% RSLogix 500 project UNTITLED_BAK061.RSS, saved by version 8.10.00.18 %
PROJECT "UNTITLED"    % processor: MicroLogix 1200 %

PROGRAM FILES
  LAD 2   19 rungs

DATA FILES
  O0 OUTPUT  4 elements
  I1 INPUT  4 elements
  S2 STATUS  66 elements
  B3 BINARY  1 elements
  T4 TIMER  7 elements
  C5 COUNTER  1 elements
  R6 CONTROL  1 elements
  N7 INTEGER  1 elements

LADDER 2
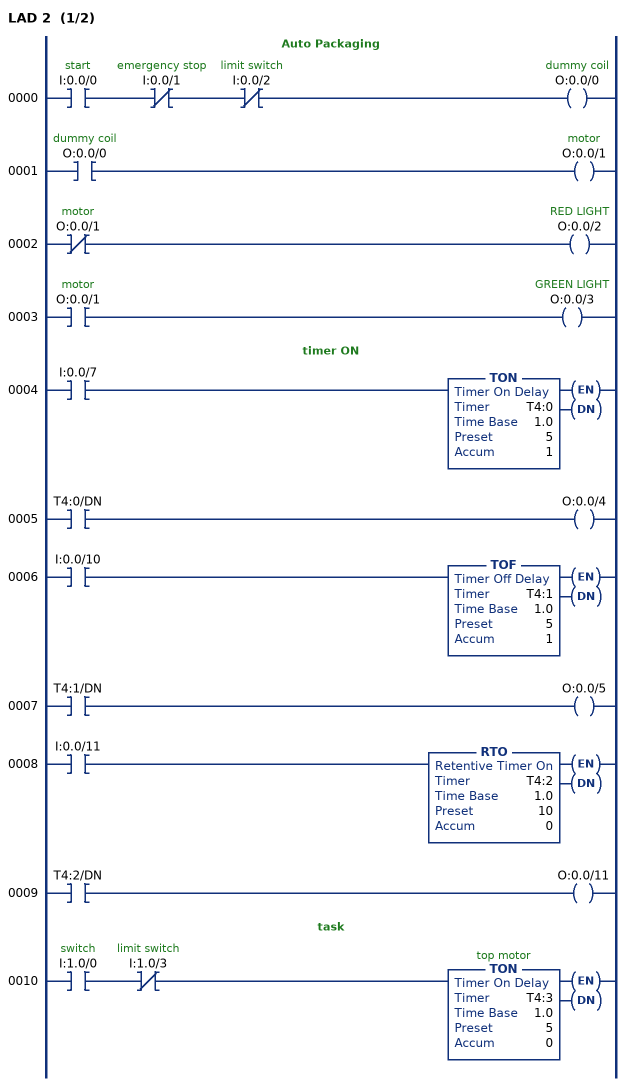
% Rung: 0 %
% TITLE: Auto Packaging %
SOR XIC I:0.0/0 XIO I:0.0/1 XIO I:0.0/2 OTE O:0.0/0 EOR
%   I:0.0/0  "start" %
%   I:0.0/1  "emergency stop" %
%   I:0.0/2  "limit switch" %
%   O:0.0/0  "dummy coil" %
% Rung: 1 %
SOR XIC O:0.0/0 OTE O:0.0/1 EOR
%   O:0.0/0  "dummy coil" %
%   O:0.0/1  "motor" %
% Rung: 2 %
SOR XIO O:0.0/1 OTE O:0.0/2 EOR
%   O:0.0/1  "motor" %
%   O:0.0/2  "RED LIGHT" %
% Rung: 3 %
SOR XIC O:0.0/1 OTE O:0.0/3 EOR
%   O:0.0/1  "motor" %
%   O:0.0/3  "GREEN LIGHT" %
% Rung: 4 %
% TITLE: timer ON %
SOR XIC I:0.0/7 TON T4:0 1.0 5 1 EOR
% Rung: 5 %
SOR XIC T4:0/DN OTE O:0.0/4 EOR
% Rung: 6 %
SOR XIC I:0.0/10 TOF T4:1 1.0 5 1 EOR
% Rung: 7 %
SOR XIC T4:1/DN OTE O:0.0/5 EOR
% Rung: 8 %
SOR XIC I:0.0/11 RTO T4:2 1.0 10 0 EOR
% Rung: 9 %
SOR XIC T4:2/DN OTE O:0.0/11 EOR
% Rung: 10 %  % edit flag set %
% TITLE: task %
SOR XIC I:1.0/0 XIO I:1.0/3 TON T4:3 1.0 5 0 EOR
%   I:1.0/0  "switch" %
%   I:1.0/3  "limit switch" %
%   T4:3  "top motor" %

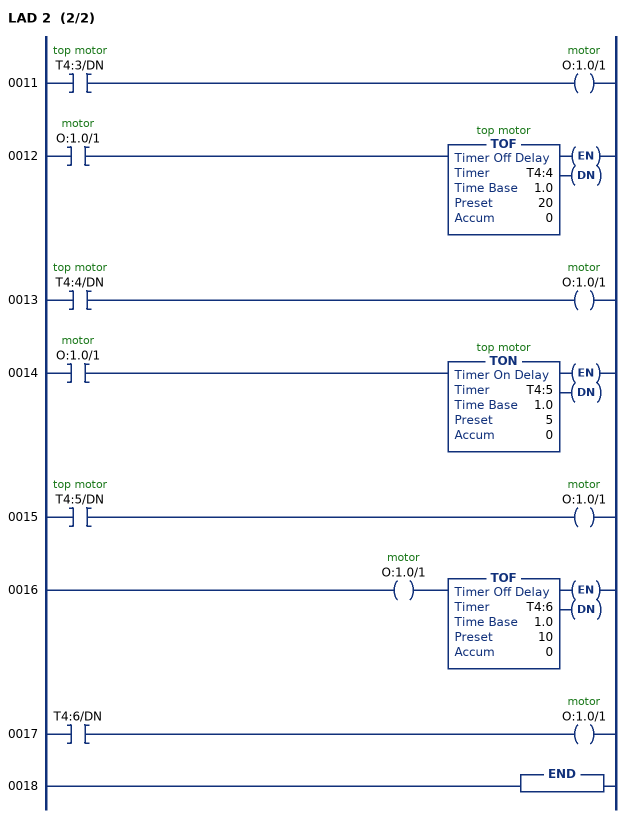
% Rung: 11 %  % edit flag set %
SOR XIC T4:3/DN OTE O:1.0/1 EOR
%   T4:3/DN  "top motor" %
%   O:1.0/1  "motor" %
% Rung: 12 %  % edit flag set %
SOR XIC O:1.0/1 TOF T4:4 1.0 20 0 EOR
%   O:1.0/1  "motor" %
%   T4:4  "top motor" %
% Rung: 13 %  % edit flag set %
SOR XIC T4:4/DN OTE O:1.0/1 EOR
%   T4:4/DN  "top motor" %
%   O:1.0/1  "motor" %
% Rung: 14 %  % edit flag set %
SOR XIC O:1.0/1 TON T4:5 1.0 5 0 EOR
%   O:1.0/1  "motor" %
%   T4:5  "top motor" %
% Rung: 15 %  % edit flag set %
SOR XIC T4:5/DN OTE O:1.0/1 EOR
%   T4:5  "top motor" %
%   O:1.0/1  "motor" %
% Rung: 16 %  % edit flag set %
SOR OTE O:1.0/1 TOF T4:6 1.0 10 0 EOR
%   O:1.0/1  "motor" %
% Rung: 17 %  % edit flag set %
SOR XIC T4:6/DN OTE O:1.0/1 EOR
%   O:1.0/1  "motor" %
% Rung: 18 %
SOR END EOR

OTHER DOCUMENTED ADDRESSES
  I:1.0/1  "limit switch"

DATA TABLE (non-zero values as saved)
DATA T4
% .PRE .ACC %
% T4:0 % 5 1
% T4:1 % 5 1
% T4:2 % 10 0
% T4:3 % 5 0
% T4:4 % 20 0
% T4:5 % 5 0
% T4:6 % 10 0
